PROGRAM Common_Pulses
VAR
	Timer_0_1_s: TON;
	Timer_1_0_s: TON;
	Timer_1_0_m: TON;
	Timer_10_0_m: TON;
	Timer0_5_s : TON;
END_VAR

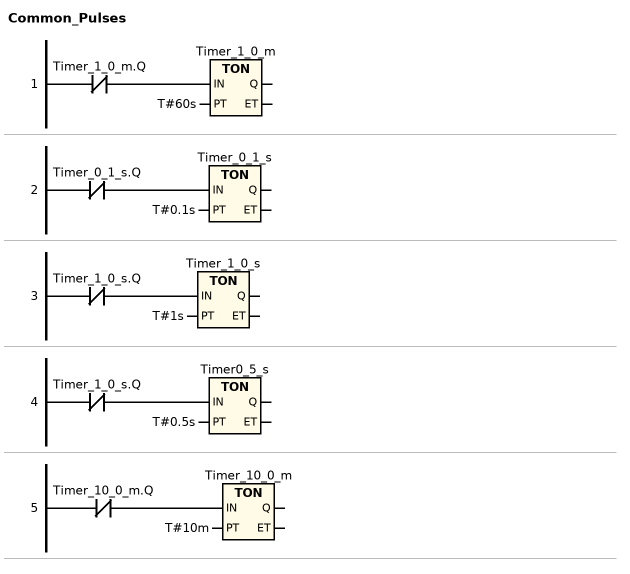
// NETWORK 1
Timer_1_0_m(IN := NOT Timer_1_0_m.Q, PT := T#60s); // TON

// NETWORK 2
Timer_0_1_s(IN := NOT Timer_0_1_s.Q, PT := T#0.1s); // TON

// NETWORK 3
Timer_1_0_s(IN := NOT Timer_1_0_s.Q, PT := T#1s); // TON

// NETWORK 4
Timer0_5_s(IN := NOT Timer_1_0_s.Q, PT := T#0.5s); // TON

// NETWORK 5
Timer_10_0_m(IN := NOT Timer_10_0_m.Q, PT := T#10m); // TON

END_PROGRAM

(* stored: Version 1.1.0.1, ProductVersion 3.1.4024.13
   POU Common_Pulses: Id {5940de78-d663-4b56-86bd-277f0a1b9c72}, SpecialFunc None *)
